// TIA Portal V17 export
// export: Created 2025-06-26T06:49:09.5921755Z, ExportSetting WithDefaults, DisplayName Totally Integrated Automation Portal, DisplayVersion V17 Update 8, DisplayName TIA Portal Openness, DisplayVersion V17 Update 8, DisplayName TIA Portal Version Control Interface, DisplayVersion V17, DisplayName STEP 7 Professional, DisplayVersion V17 Update 8, DisplayName STEP 7 Safety, DisplayVersion V17 Update 6, DisplayName WinCC Advanced, DisplayVersion V17 Update 8
FUNCTION_BLOCK "InputProcessing"   // FB48, FBD
{ S7_Optimized_Access := 'TRUE' }
AUTHOR : Heaten
VERSION : 0.1
// stored: AutoNumber true, IsIECCheckEnabled false, IsRetainMemResEnabled false, MemoryReserve 0, SetENOAutomatically false, UDAEnableTagReadback false
   VAR
      AnalogInputProcessing_DB { ExternalAccessible := 'False'; ExternalVisible := 'False'; ExternalWritable := 'False'} : "AnalogInputProcessing";
      InputAlarmHandling_DB { ExternalAccessible := 'False'; ExternalVisible := 'False'; ExternalWritable := 'False'} : "InputAlarmHandling";
      InverterDriveProcessing_DB : "InverterDriveProcessing";
      DigitalInputProcessing_DB { ExternalAccessible := 'False'; ExternalVisible := 'False'; ExternalWritable := 'False'} : "DigitalInputProcessing";
      Simulation_DB { ExternalAccessible := 'False'; ExternalVisible := 'False'; ExternalWritable := 'False'} : "Simulation";
      HBL_HV_640 { S7_SetPoint := 'True'} : "fbProcessValve2_V2";
      HBL_HV_670 { S7_SetPoint := 'True'} : "fbProcessValve2_V2";
      CPC_HV_852 { S7_SetPoint := 'True'} : "fbProcessValve2_V2";
      HBL_HV_861 { S7_SetPoint := 'True'} : "fbProcessValve2_V2";
      bTempOpenReq { S7_SetPoint := 'True'} : Bool;
      bTempCloseReq : Bool;
      bTempOpenStat : Bool;
      bTempCloseStat : Bool;
   END_VAR
BEGIN

REGION Network 1: Digital inputs
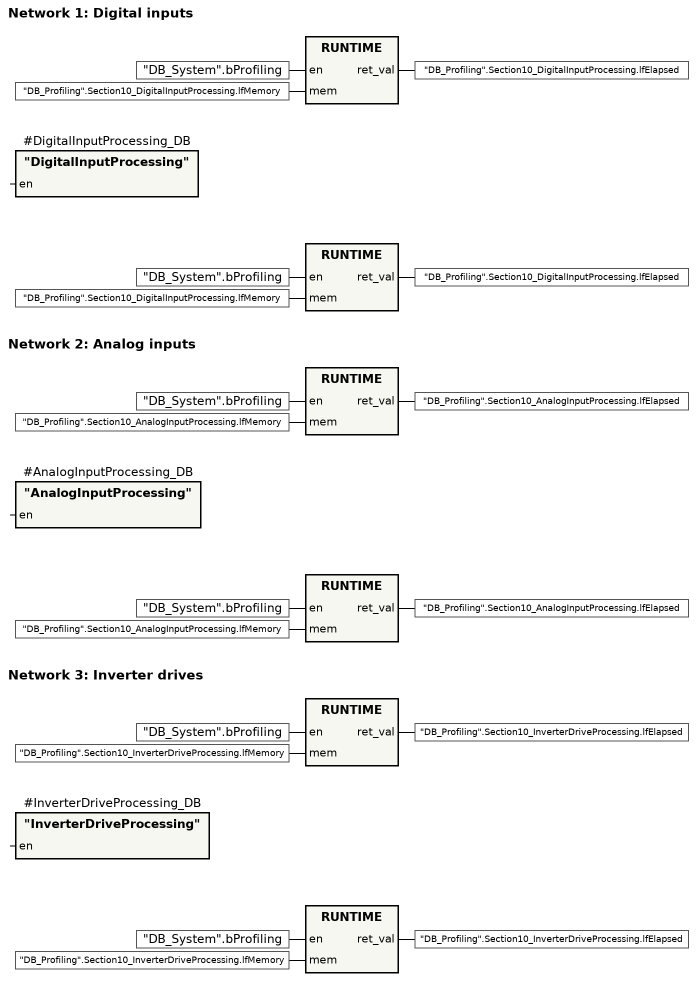
   // no SCL statement known for Runtime: written as a call
   IF "DB_System".bProfiling THEN
       "DB_Profiling".Section10_DigitalInputProcessing.lfElapsed := Runtime(mem := "DB_Profiling".Section10_DigitalInputProcessing.lfMemory);
   END_IF;
   #DigitalInputProcessing_DB();   // "DigitalInputProcessing"
   IF "DB_System".bProfiling THEN
       "DB_Profiling".Section10_DigitalInputProcessing.lfElapsed := Runtime(mem := "DB_Profiling".Section10_DigitalInputProcessing.lfMemory);
   END_IF;
END_REGION

REGION Network 2: Analog inputs
   // no SCL statement known for Runtime: written as a call
   IF "DB_System".bProfiling THEN
       "DB_Profiling".Section10_AnalogInputProcessing.lfElapsed := Runtime(mem := "DB_Profiling".Section10_AnalogInputProcessing.lfMemory);
   END_IF;
   #AnalogInputProcessing_DB();   // "AnalogInputProcessing"
   IF "DB_System".bProfiling THEN
       "DB_Profiling".Section10_AnalogInputProcessing.lfElapsed := Runtime(mem := "DB_Profiling".Section10_AnalogInputProcessing.lfMemory);
   END_IF;
END_REGION

REGION Network 3: Inverter drives
   // no SCL statement known for Runtime: written as a call
   IF "DB_System".bProfiling THEN
       "DB_Profiling".Section10_InverterDriveProcessing.lfElapsed := Runtime(mem := "DB_Profiling".Section10_InverterDriveProcessing.lfMemory);
   END_IF;
   #InverterDriveProcessing_DB();   // "InverterDriveProcessing"
   IF "DB_System".bProfiling THEN
       "DB_Profiling".Section10_InverterDriveProcessing.lfElapsed := Runtime(mem := "DB_Profiling".Section10_InverterDriveProcessing.lfMemory);
   END_IF;
END_REGION

REGION Network 4: Process valves
   // Own FB?
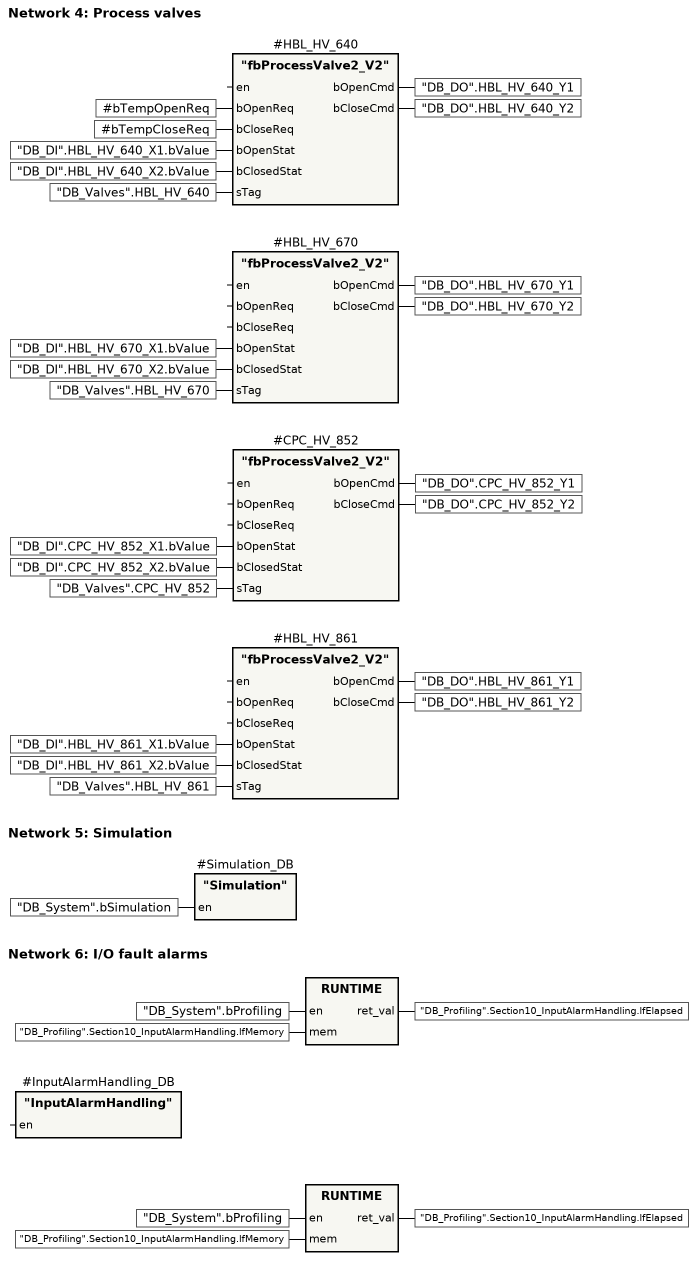
   #HBL_HV_640(bOpenReq := #bTempOpenReq,   // "fbProcessValve2_V2"
               bCloseReq := #bTempCloseReq,
               bOpenStat := "DB_DI".HBL_HV_640_X1.bValue,
               bClosedStat := "DB_DI".HBL_HV_640_X2.bValue,
               sTag := "DB_Valves".HBL_HV_640,
               bOpenCmd => "DB_DO".HBL_HV_640_Y1,
               bCloseCmd => "DB_DO".HBL_HV_640_Y2);
   #HBL_HV_670(bOpenStat := "DB_DI".HBL_HV_670_X1.bValue,   // "fbProcessValve2_V2"
               bClosedStat := "DB_DI".HBL_HV_670_X2.bValue,
               sTag := "DB_Valves".HBL_HV_670,
               bOpenCmd => "DB_DO".HBL_HV_670_Y1,
               bCloseCmd => "DB_DO".HBL_HV_670_Y2);
   #CPC_HV_852(bOpenStat := "DB_DI".CPC_HV_852_X1.bValue,   // "fbProcessValve2_V2"
               bClosedStat := "DB_DI".CPC_HV_852_X2.bValue,
               sTag := "DB_Valves".CPC_HV_852,
               bOpenCmd => "DB_DO".CPC_HV_852_Y1,
               bCloseCmd => "DB_DO".CPC_HV_852_Y2);
   #HBL_HV_861(bOpenStat := "DB_DI".HBL_HV_861_X1.bValue,   // "fbProcessValve2_V2"
               bClosedStat := "DB_DI".HBL_HV_861_X2.bValue,
               sTag := "DB_Valves".HBL_HV_861,
               bOpenCmd => "DB_DO".HBL_HV_861_Y1,
               bCloseCmd => "DB_DO".HBL_HV_861_Y2);
END_REGION

REGION Network 5: Simulation
   IF "DB_System".bSimulation THEN
       #Simulation_DB();   // "Simulation"
   END_IF;
END_REGION

REGION Network 6: I/O fault alarms
   // Put this last so that any Simulation code doesn't have to fix up any alarms
   // no SCL statement known for Runtime: written as a call
   IF "DB_System".bProfiling THEN
       "DB_Profiling".Section10_InputAlarmHandling.lfElapsed := Runtime(mem := "DB_Profiling".Section10_InputAlarmHandling.lfMemory);
   END_IF;
   #InputAlarmHandling_DB();   // "InputAlarmHandling"
   IF "DB_System".bProfiling THEN
       "DB_Profiling".Section10_InputAlarmHandling.lfElapsed := Runtime(mem := "DB_Profiling".Section10_InputAlarmHandling.lfMemory);
   END_IF;
END_REGION
END_FUNCTION_BLOCK
